FUNCTION_BLOCK FB_PressureSensor
VAR_INPUT
END_VAR
VAR_OUTPUT
END_VAR
VAR
	rPressure : REAL;
END_VAR

PROPERTY getPressure : REAL
GET
getPressure := rPressure;
END_GET
END_PROPERTY

END_FUNCTION_BLOCK

(* stored: Version 1.1.0.1, ProductVersion 3.1.4024.11
   POU FB_PressureSensor: Id {17567b52-9a99-4ecd-ac02-8e7eeae25c38}, SpecialFunc None
   Property getPressure: Id {a745bce9-e7b1-4e02-b18e-265bce1f8258}
   Get Get: Id {d653a4e6-8290-4a1d-af67-b1bc9a168e9b} *)
